// TIA Portal V19 export
DATA_BLOCK "Com_ToPolygonFiller"   // DB472
{ S7_Optimized_Access := 'TRUE' }
// stored: AutoNumber false, MemoryReserve 0
   VAR RETAIN
      CIP : Struct   // CIP Signals From APV AHV
         LifeBit : Bool;   // Process_LifeBit
         SpareBool_0_1 : Bool;
         SpareBool_0_2 : Bool;
         SpareBool_0_3 : Bool;
         SpareBool_0_4 : Bool;
         SpareBool_0_5 : Bool;
         SpareBool_0_6 : Bool;
         SpareBool_0_7 : Bool;
         ReadyForCIP : Bool;   // Process_ReadyForCIP
         NoTimeStop : Bool;   // Process_NoTimeStop
         ReleaseCIPReturnPump : Bool;   // Process_ReleaseCIPReturnPump
         CIPStepRelease : Bool;   // Process_CIPStepRelease
         CIPRunningF1 : Bool;   // Process_CIPRunning (Optional)
         FlippingOfSeatF1 : Bool;   // Process_FlippingOfSeat (Optional)
         CIPRunningF2 : Bool;
         FlippingOfSeatF2 : Bool;
         SpareBool_2_0 : Bool;
         SpareBool_2_1 : Bool;
         SpareBool_2_2 : Bool;
         SpareBool_2_3 : Bool;
         SpareBool_2_4 : Bool;
         SpareBool_2_5 : Bool;
         SpareBool_2_6 : Bool;
         SpareBool_2_7 : Bool;
         SpareBool_3_0 : Bool;
         SpareBool_3_1 : Bool;
         SpareBool_3_2 : Bool;
         SpareBool_3_3 : Bool;
         SpareBool_3_4 : Bool;
         SpareBool_3_5 : Bool;
         SpareBool_3_6 : Bool;
         SpareBool_3_7 : Bool;
         Spacer : Array[0..11] of Word;
      END_STRUCT;
      SIP : Struct   // Sterilisation Signals from Hassia
         Release : Bool;   // Process_SIPRelease
         LineSterileFiller1 : Bool;   // Process_LineSterileFiller1
         LineSterileFiller2 : Bool;   // Process_LineSterileFiller2
         SIPLineRunningF1 : Bool;   // Process_SIPLineRunning from Fruit Plant Alsafe
         SIPLineRunningF2 : Bool;   // Process_SIPLineRunning from APV AHV
         spacer : Array[0..12] of Word;
      END_STRUCT;
      Production : Struct   // Production Signals from Hassia
         ReadyFiller1 : Bool;   // Process_ProductReadyFiller1
         ReadyFiller2 : Bool;   // Process_ProductReadyFiller2
         SpareBool_0_2 : Bool;   // spare
         SpareBool_0_3 : Bool;   // spare
         int_2 : Int;   // spare
         Int_4 : Int;   // spare
         Spacer : Array[0..10] of Word;   // spare
      END_STRUCT;
   END_VAR
BEGIN
END_DATA_BLOCK
